FUNCTION_BLOCK FB_SlaveArmCtrlCycleTest EXTENDS FB_SlaveArmCtrlBase
VAR_INPUT
END_VAR
VAR_OUTPUT
END_VAR
VAR
	//arm id
	m_armId:INT;			
	
	//test step
	m_testStep:INT:=-1;
	
	//DH joint position	
	m_homeDHJntPos,m_startDHJntPos,m_endDHJntPos:Vec6d;
	
	//startJntPos,endJntPos :Vec8d;
	m_initJntPos,m_startJntPos,m_endJntPos :Vec8d;
	
	//motion parameters
	m_maxjntVel,m_maxjntAcc,m_maxjntJerk:Vec8d;
	
	//time
	m_time:LREAL;
		
	//test point
	m_testPoint:INT;
	
	//motion start
	m_startMotion:BOOL;
	m_startMotionLast:BOOL;
	
	//joint position gap
	m_jntDist:Vec6d:=[30.0*g_deg2Rad,30.0*g_deg2Rad,0.030,30.0*g_deg2Rad,30.0*g_deg2Rad,30.0*g_deg2Rad];	
	
	//Trajectory planner
	m_Planner: FB_TrajMoveJ;
END_VAR

// override this function in each exact controller
METHOD PROTECTED calcCmdJntPos : BOOL
VAR_IN_OUT CONSTANT
	// endoscope pose in cart coordinate
	i_endoscopePose : ST_Frame;
	
	// master arm data
	i_masterStatus :ST_MasterStatus;
	
	// setup arm data
	i_setupStatus: ST_SetupStatus;
	
	// slave arm data
	i_slaveArm :FB_SlaveArm;
END_VAR


//init parameters flag
m_startMotion:=gvl_testCycle.g_startMotion[m_armId];
IF (m_startMotionLast=FALSE) AND (m_startMotion=TRUE)THEN
	m_testStep:=0;
END_IF
m_startMotionLast:=m_startMotion;

//frequency test and step test
testMotion(i_slaveArm);

//update the information
updateInfo(i_slaveArm);
END_METHOD

// override this function in each exact controller
// NOTICE: set joint control mode here, and do some initialization if needed
METHOD PUBLIC init : BOOL
VAR_IN_OUT CONSTANT
	i_slaveArm	:FB_SlaveArm;
END_VAR
VAR_IN_OUT 
	r_slaveArmCtrlCmd :ST_SlaveArmCtrlCmds;
END_VAR

VAR
	i:INT;
END_VAR


SUPER^.Init(i_slaveArm,r_slaveArmCtrlCmd);

//variable initialization
m_armId:=i_slaveArm.armIdx;

//target DH joint position
m_homeDHJntPos:=gvl_accuracyTest.g_originJntPos;
FOR i:=1 TO 6 BY 1 DO
	m_homeDHJntPos[i]:=i_slaveArm.curDHJntPos[i];
	//m_jntDist[i]:=(GVL_SlaveMotorParameters.g_maxJntPos[i]-GVL_SlaveMotorParameters.g_minJntPos[i])*0.1;
	m_startDHJntPos[i]:=m_homeDHJntPos[i]-m_jntDist[i];
	m_endDHJntPos[i]:=m_homeDHJntPos[i]+m_jntDist[i];
END_FOR

//start flag
m_startMotionLast:=FALSE;

//velocity---acceleration---jerk
vecMultiNum(GVL_SlaveMotorParameters.g_maxJntVel,0.2,m_maxjntVel);
vecMultiNum(m_maxjntVel,3,m_maxjntAcc);
vecMultiNum(m_maxjntAcc,3,m_maxjntJerk);
END_METHOD

METHOD testMotion : BOOL
VAR_INPUT
	// slave arm data
	i_slaveArm :FB_SlaveArm;
END_VAR

VAR
	homeDHPos,startDHPos,endDHPos :Vec6d;
END_VAR

CASE m_testStep OF
	0: //init
		m_testPoint:=1;		
		m_testStep:=10;
		
		
	10: //Trajectory parameter initialization
		startDHPos:=i_slaveArm.curDHJntPos;
		IF (m_testPoint=1) THEN
			endDHPos:=m_startDHJntPos;
		ELSIF (m_testPoint=2) THEN
			endDHPos:=m_homeDHJntPos;
		ELSIF (m_testPoint=3) THEN
			endDHPos:=m_endDHJntPos;
		END_IF
		i_slaveArm.instrument.instruIK(startDHPos,0, o_jntPos=>m_startJntPos);
		i_slaveArm.instrument.instruIK(endDHPos,0, o_jntPos=>m_endJntPos);
		
		m_Planner.init(i_startJntPos:= m_startJntPos, 	i_targetJntPos:= m_endJntPos, 	i_maxJntVel:= m_maxjntVel, 	i_maxJntAcc:= m_maxjntAcc, 	i_maxJntJerk:= m_maxjntJerk);
		IF (m_Planner.isGene=FALSE) THEN
			m_testStep:=30;
		ELSE
			m_time:=0; m_testStep:=20;
		END_IF
		
		
	20: //start motion
		m_time:=m_time+g_slaveArmCtrlCycleTime;
		m_Planner.evaluate(t:= m_time, jntPos=> m_cmdJntPos, jntVel=> m_cmdJntVel, jntAcc=> m_cmdJntAcc);
		
		IF (m_time>m_Planner.duration) THEN
			m_testStep:=10;			
			m_testPoint:=m_testPoint+1;
			IF (m_testPoint>3) THEN
				m_testPoint:=1;
			END_IF
		END_IF		
		
		//end the motion
		IF (m_startMotion=FALSE) THEN
			m_testStep:=30;
		END_IF
		
		
	30: //end the motion
		m_testStep:=-1;		
END_CASE
END_METHOD

METHOD updateInfo : BOOL
VAR_INPUT
	// slave arm data
	i_slaveArm :FB_SlaveArm;
END_VAR

VAR
	i:INT;
END_VAR


FOR i:=1 TO g_sJntNum BY 1 DO
	gvl_TestCycle.g_slaveArmMotorEncoder[m_armId][i]:=i_slaveArm.m_joints[i].m_motorInputs.m_motorEncoder;
	gvl_TestCycle.g_slaveArmjntEncoder[m_armId][i]:=i_slaveArm.m_joints[i].m_motorInputs.m_linkEncoder;
END_FOR
END_METHOD

END_FUNCTION_BLOCK

(* stored: Version 1.1.0.1, ProductVersion 3.1.4024.11
   POU FB_SlaveArmCtrlCycleTest: Id {81d205fb-0875-4a86-a828-a1e7ff543989}, SpecialFunc None
   Method calcCmdJntPos: Id {e765b525-c56e-4df7-9941-bd0b34c07d3f}
   Method init: Id {a68df1fd-fda0-4f57-b897-de892ee6d53d}
   Method testMotion: Id {19b26b72-892d-4dd3-8aad-e8216d36cbf9}
   Method updateInfo: Id {2c3bedc5-efa1-409d-9953-1b6bffd89a98} *)
